FUNCTION_BLOCK L2_StateTracker (* Basic Function Block Type *)
  (* Standard: 61499-2 *)
  (* Version 0.0, 2014-12-04, EQUEROL, UJI *)
  (* Version 1.0, 2016-01-18, EQUEROL, UJI *)
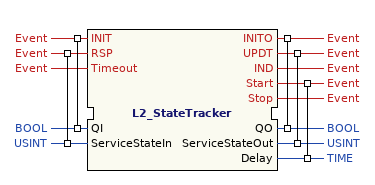
  EVENT_INPUT
    INIT WITH QI; (* Initialize keep alive service *)
    RSP WITH ServiceStateIn; (* Service state request response *)
    Timeout; (* Delay timeout *)
  END_EVENT
  EVENT_OUTPUT
    INITO WITH QO; (* Initialization confirmation *)
    UPDT WITH ServiceStateOut; (* Update Machine state *)
    IND; (* Request machine service state *)
    Start WITH Delay; (* Timeout start *)
    Stop; (* Timeout stop *)
  END_EVENT
  VAR_INPUT
    QI : BOOL; (* Input event qualifier *)
    ServiceStateIn : USINT; (* Machine service state *)
  END_VAR
  VAR_OUTPUT
    QO : BOOL; (* Output event qualifier *)
    ServiceStateOut : USINT; (* Machine service state *)
    Delay : TIME; (* Timeout delay *)
  END_VAR
  VAR
    TOCounter : USINT := 0; (* Timeouts counter *)
    MaxTO : USINT := 10; (* Maximum number fo timeouts *)
  END_VAR
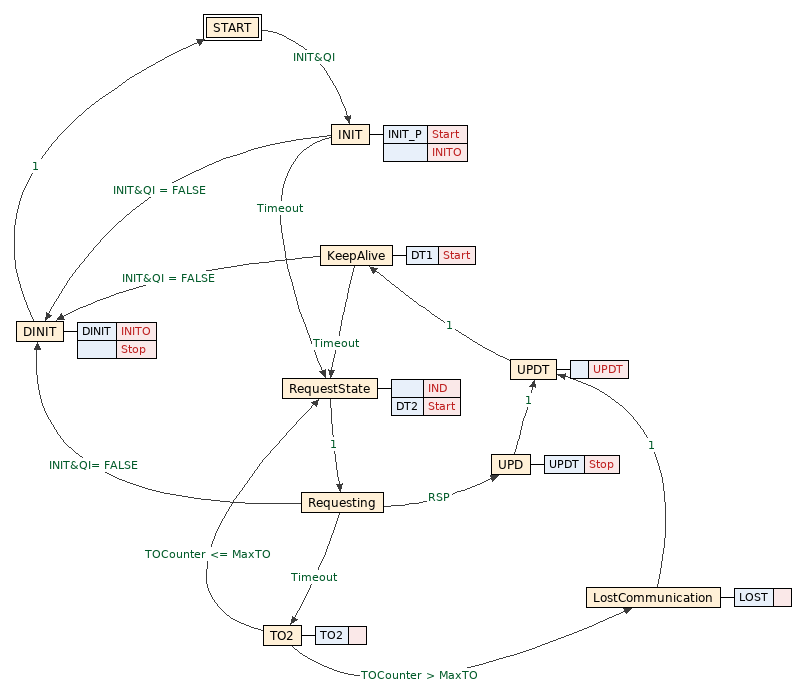
  EC_STATES
    START; (* Initial State *)
    DINIT : DINIT -> INITO, -> Stop; (* Initialization *)
    UPDT : -> UPDT; (* Normal execution *)
    UPD : UPDT -> Stop;
    RequestState : -> IND, DT2 -> Start;
    KeepAlive : DT1 -> Start;
    Requesting;
    TO2 : TO2;
    LostCommunication : LOST;
    INIT : INIT_P -> Start, -> INITO;
  END_STATES
  EC_TRANSITIONS
    UPD TO UPDT := 1;
    RequestState TO Requesting := 1;
    KeepAlive TO RequestState := Timeout;
    Requesting TO UPD := RSP;
    UPDT TO KeepAlive := 1;
    Requesting TO TO2 := Timeout;
    TO2 TO RequestState := TOCounter <= MaxTO;
    TO2 TO LostCommunication := TOCounter > MaxTO;
    LostCommunication TO UPDT := 1;
    KeepAlive TO DINIT := INIT&QI = FALSE;
    Requesting TO DINIT := INIT&QI= FALSE;
    START TO INIT := INIT&QI;
    INIT TO RequestState := Timeout;
    DINIT TO START := 1;
    INIT TO DINIT := INIT&QI = FALSE;
  END_TRANSITIONS
  ALGORITHM INIT_P IN ST: (* Initialization algorithm *)
QO := TRUE;
Delay := TIME#2000ms;
  END_ALGORITHM
  ALGORITHM UPDT IN ST: (* Update service state algo *)
ServiceStateOut := ServiceStateIn;
(*Reset timeouts counter*)
TOCounter := 0;
  END_ALGORITHM
  ALGORITHM DT1 IN ST: (* Keep alive algo *)
(*Periodic machine check*)
Delay := TIME#60000ms;
  END_ALGORITHM
  ALGORITHM DT2 IN ST: (* REQS algo *)
(*A Machine is expected to answer within a second to a request state event*)
Delay := TIME#1000ms;
  END_ALGORITHM
  ALGORITHM TO2 IN ST: (* Algorithm to control the number fo timeouts while requesting the service state *)
TOCounter := TOCounter + 1;
  END_ALGORITHM
  ALGORITHM LOST IN ST: (* lost communication algo *)
(*We lost the communication with the Machine service*)
ServiceStateOut :=  0;
  END_ALGORITHM
  ALGORITHM DINIT IN ST: (* new algorithm *)
QO := FALSE;
  END_ALGORITHM
END_FUNCTION_BLOCK
